SUBAPPLICATION ZylinderSingle (* Single actuated zylinder where the home position is automatically reached with a spring *)
  (* Standard: 61499-2 *)
  (* Version 1.0, 2018-07-10, az *)
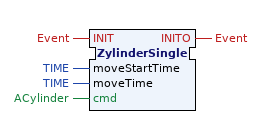
  EVENT_INPUT
    INIT;
  END_EVENT
  EVENT_OUTPUT
    INITO;
  END_EVENT
  VAR_INPUT
    moveStartTime : TIME;
    moveTime : TIME;
  END_VAR
  SOCKETS
    cmd : ACylinder;
  END_SOCKETS
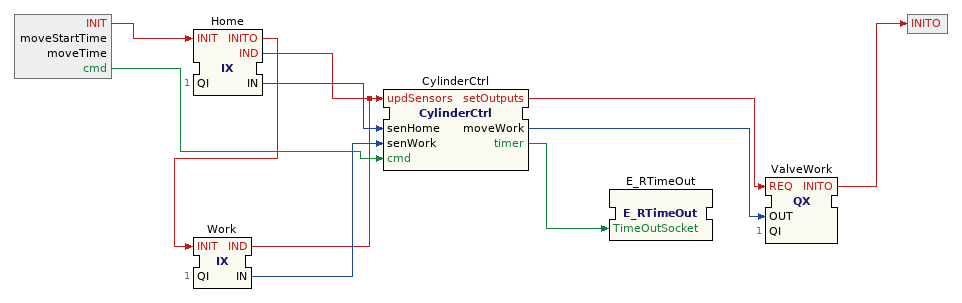
  FBS
    ValveWork : QX(QI := 1);
    Home : IX(QI := 1);
    Work : IX(QI := 1);
    E_RTimeOut : E_RTimeOut;
    CylinderCtrl : CylinderCtrl;
  END_FBS
  EVENT_CONNECTIONS
    Home.INITO TO Work.INIT;
    INIT TO Home.INIT;
    ValveWork.INITO TO INITO;
    Home.IND TO CylinderCtrl.updSensors;
    Work.IND TO CylinderCtrl.updSensors;
    CylinderCtrl.setOutputs TO ValveWork.REQ;
  END_CONNECTIONS
  DATA_CONNECTIONS
    Home.IN TO CylinderCtrl.senHome;
    Work.IN TO CylinderCtrl.senWork;
    CylinderCtrl.moveWork TO ValveWork.OUT;
  END_CONNECTIONS
  ADAPTER_CONNECTIONS
    CylinderCtrl.timer TO E_RTimeOut.TimeOutSocket;
    cmd TO CylinderCtrl.cmd;
  END_CONNECTIONS
END_SUBAPPLICATION
